{attribute addProperty BoxType "EK1960-2600-0021"}
{attribute addProperty Id "Module_1_FSoEModule_1_FSoE_1C2EAE46240300Module_2_FSOUTModule_2_FSOUT_3AD10D8E224280Module_3_FSLOGICModule_3_FSLOGIC_3E6251391620WcStateAT %I*WcState_DC9C971540.50InfoDataAT %I*InfoData_BC63D37F80100"}
{attribute addProperty CRC "2592253150"}
{attribute addProperty SizeInBites "564"}
{attribute addProperty SizeInBytes "70.5"}
TYPE EK1960_3617E9AF :
STRUCT
	{attribute addProperty Name "Module_1_FSoE"}
	Module_1_FSoE : Module_1_FSoE_1C2EAE46;
	{attribute addProperty Name "Module_2_FSOUT"}
	Module_2_FSOUT : Module_2_FSOUT_3AD10D8E;
	{attribute addProperty Name "Module_3_FSLOGIC"}
	Module_3_FSLOGIC : Module_3_FSLOGIC_3E625139;
	{attribute addProperty Name "WcState"}
	WcState : WcState_DC9C9715;
	{attribute addProperty Name "InfoData"}
	InfoData : InfoData_BC63D37F;
END_STRUCT
END_TYPE

(* stored: Version 1.2.0.0, ProductVersion 3.1.4024.9
   DUT EK1960_3617E9AF: Id {d2ef520a-9d8b-4946-9f2a-45879d3c8f2c} *)
